// TwinCAT 3 PLC project Untitled1
// ProgramVersion: 3.1.4023.0
// libraries:
//   PLCToolbox, * (Beckhoff Automation LLC.)
//   Tc2_Standard, * (Beckhoff Automation GmbH)
//   Tc2_System, * (Beckhoff Automation GmbH)
//   Tc3_Module, * (Beckhoff Automation GmbH)
// project tree:
//   / PlcTask.TcTTO
//   POUs/ MAIN.TcPOU
// real-time tasks:
//   TASK PlcTask: cycle T#10ms, priority 20, ADS port 350

CONFIGURATION Untitled1
    RESOURCE PLC ON TwinCAT3
        TASK PlcTask(INTERVAL := T#10ms, PRIORITY := 20);
        PROGRAM MAIN WITH PlcTask : MAIN;
    END_RESOURCE
END_CONFIGURATION

// ---- POUs/MAIN.TcPOU
PROGRAM MAIN
VAR	            	
	Runnning		:BOOL;
	Light			:BOOL;
	
	Data			:FB_GenerateData;

	
	fbFlasher		:FB_Flasher;	
END_VAR


fbFlasher(
	xEnable:=Runnning , 
	tTimeOff:=T#1S , 
	tTimeOn:=T#1S , 
	tTimeTillOn=> , 
	tTimeTillOff=> , 
	xStatus=> Light);
	

Data( );

END_PROGRAM
